// TIA Portal V19 export
TYPE "LAF_typeNgConveyorEm1Parameters"
// stored: Access Published
   STRUCT
      cm2Axis111 : "LAF_typeAxisParameters";
      cm3NgStrap : "LAF_typeNgStrapParameters";
   END_STRUCT;
END_TYPE
